(* IEC 61131-3 sources: pandora/pandora/aws-platform-main/aws-platform-main/test/Api, 3 files *)

(* ---- IoGroups.st ---- *)
USING AxUnit;

NAMESPACE Esab.Api.Test

    {TestFixture}
    CLASS DigitalOutputGroupTests
        VAR PRIVATE
            output : DigitalOutputGroup;
        END_VAR

        {FixtureSetup}
        METHOD PUBLIC TestFixtureSetup
            ;
        END_METHOD

        {TestSetup}
        METHOD PUBLIC TestSetup
            output.Output.Reset();
            output.Value := FALSE;
        END_METHOD

        {Test}
        METHOD PUBLIC MyTestMethod
            output.Output.Set();
            Assert.Equal(output.Value, FALSE);
            output.Write();
            Assert.Equal(output.Value, TRUE);

            output.Output.Reset();
            Assert.Equal(output.Value, TRUE);
            output.Write();
            Assert.Equal(output.Value, FALSE);
        END_METHOD
    END_CLASS

END_NAMESPACE

(* ---- WebApi.st ---- *)
USING Esab.Utils;
USING Esab.WeldSystem.PowerSources.Mock;
USING Esab.WeldSystem.PowerSources;
USING Esab.Motion.Mock;
USING Esab.Utils.Alarming.Mock;
USING Esab.Utils.Assets.Mock;
USING Esab.Utils.Assets;

USING AxUnit;

NAMESPACE Esab.Api.Test

    {TestFixture}
    {Category(WebApi)}
    CLASS WebApiSlideCrossTests
        VAR PRIVATE
            _api : WebApi;
            _defaultApi : WebApi;
            _webApiData : WebApiData;
            _defaultWebApiData : WebApiData;
            _horizontalSlideMock : ToPosAxisMock;
            _verticalSlideMock : ToPosAxisMock;
            _assetsManagerMock : AssetsManagerMock;
        END_VAR

        {FixtureSetup}
        METHOD PUBLIC TestFixtureSetup
            _api := _defaultApi;
            _api.Setup(_assetsManagerMock, REF(_webApiData));
        END_METHOD

        {TestSetup}
        METHOD PUBLIC TestSetup
            _webApiData := _defaultWebApiData;

            _horizontalSlideMock.MockReset();
            _verticalSlideMock.MockReset();
            _assetsManagerMock.MockReset();

            // Configure assets manager mock: by default hand out the horizontal axis when requested
            _assetsManagerMock.RequestAssetHandleMock.Qualifier := AssetIdentifier#HorizontalSlideAxis;
            _assetsManagerMock.RequestAssetHandleMock.Asset := REF(_horizontalSlideMock);
            // Observables are not required for these tests; let ObserveAsset return NULL by default
            _assetsManagerMock.ObserveAssetMock.Value := NULL;
        END_METHOD

        {Test}
        METHOD PUBLIC HorizontalSlideEnable
            _webApiData.Inputs.HorizontalSlide.Commands.Enable.Execute.Read(TRUE);

            _api.Execute();

            Assert.Equal(_horizontalSlideMock.PowerOnMock.GetCallCount(), UINT#1);
        END_METHOD

        {Test}
        METHOD PUBLIC VerticalSlideEnable
            // Reconfigure assets manager mock to return vertical axis for this test
            _assetsManagerMock.RequestAssetHandleMock.Qualifier := AssetIdentifier#VerticalSlideAxis;
            _assetsManagerMock.RequestAssetHandleMock.Asset := REF(_verticalSlideMock);

            _webApiData.Inputs.VerticalSlide.Commands.Enable.Execute.Read(TRUE);

            _api.Execute();

            Assert.Equal(_verticalSlideMock.PowerOnMock.GetCallCount(), UINT#1);
        END_METHOD

        {Test}
        METHOD PUBLIC HorizontalSlideAbsolutePositionCommand
            _webApiData.Inputs.HorizontalSlide.Commands.Positioning.CommandType.Read(PositioningCommandType#Absolute);
            _webApiData.Inputs.HorizontalSlide.Commands.Positioning.Position.Read(REAL#1.0);
            _webApiData.Inputs.HorizontalSlide.Commands.Positioning.Velocity.Read(REAL#2.0);
            _webApiData.Inputs.HorizontalSlide.Commands.Positioning.Acceleration.Read(REAL#3.0);
            _webApiData.Inputs.HorizontalSlide.Commands.Positioning.Deceleration.Read(REAL#4.0);
            _webApiData.Inputs.HorizontalSlide.Commands.Positioning.Jerk.Read(REAL#5.0);
            _webApiData.Inputs.HorizontalSlide.Commands.Positioning.Execute.Read(TRUE);

            _api.Execute();

            Assert.Equal(_horizontalSlideMock.ExecutePositioningCommandMock.GetCallCount(), UINT#1);
            //Assert.Equal(_horizontalSlideHandlerMock.ExecuteCommandMock.Command.Id, 123);
            Assert.Equal(_horizontalSlideMock.ExecutePositioningCommandMock.Command.CommandType, Esab.Motion.AxisCommandType#Absolute);
            Assert.Equal(_horizontalSlideMock.ExecutePositioningCommandMock.Command.Position, 1.0);
            Assert.Equal(_horizontalSlideMock.ExecutePositioningCommandMock.Command.Velocity, 2.0);
            Assert.Equal(_horizontalSlideMock.ExecutePositioningCommandMock.Command.Acceleration, 3.0);
            Assert.Equal(_horizontalSlideMock.ExecutePositioningCommandMock.Command.Deceleration, 4.0);
            Assert.Equal(_horizontalSlideMock.ExecutePositioningCommandMock.Command.Jerk, 5.0);
            ;
        END_METHOD

        {Test}
        METHOD PUBLIC HorizontalSlideRelativePositionCommand
            _webApiData.Inputs.HorizontalSlide.Commands.Positioning.CommandType.Read(PositioningCommandType#Relative);
            _webApiData.Inputs.HorizontalSlide.Commands.Positioning.Position.Read(REAL#1.0);
            _webApiData.Inputs.HorizontalSlide.Commands.Positioning.Velocity.Read(REAL#2.0);
            _webApiData.Inputs.HorizontalSlide.Commands.Positioning.Acceleration.Read(REAL#3.0);
            _webApiData.Inputs.HorizontalSlide.Commands.Positioning.Deceleration.Read(REAL#4.0);
            _webApiData.Inputs.HorizontalSlide.Commands.Positioning.Jerk.Read(REAL#5.0);
            _webApiData.Inputs.HorizontalSlide.Commands.Positioning.Execute.Read(TRUE);

            _api.Execute();

            Assert.Equal(_horizontalSlideMock.ExecutePositioningCommandMock.GetCallCount(), UINT#1);
            //Assert.Equal(_horizontalSlideHandlerMock.ExecuteCommandMock.Command.Id, 123);
            Assert.Equal(_horizontalSlideMock.ExecutePositioningCommandMock.Command.CommandType, Esab.Motion.AxisCommandType#Relative);
            Assert.Equal(_horizontalSlideMock.ExecutePositioningCommandMock.Command.Position, 1.0);
            Assert.Equal(_horizontalSlideMock.ExecutePositioningCommandMock.Command.Velocity, 2.0);
            Assert.Equal(_horizontalSlideMock.ExecutePositioningCommandMock.Command.Acceleration, 3.0);
            Assert.Equal(_horizontalSlideMock.ExecutePositioningCommandMock.Command.Deceleration, 4.0);
            Assert.Equal(_horizontalSlideMock.ExecutePositioningCommandMock.Command.Jerk, 5.0);
        END_METHOD

        {Test}
        METHOD PUBLIC HorizontalSlideVelocityCommand
            _webApiData.Inputs.HorizontalSlide.Commands.Positioning.CommandType.Read(PositioningCommandType#Velocity);
            _webApiData.Inputs.HorizontalSlide.Commands.Positioning.Position.Read(REAL#1.0);
            _webApiData.Inputs.HorizontalSlide.Commands.Positioning.Velocity.Read(REAL#2.0);
            _webApiData.Inputs.HorizontalSlide.Commands.Positioning.Acceleration.Read(REAL#3.0);
            _webApiData.Inputs.HorizontalSlide.Commands.Positioning.Deceleration.Read(REAL#4.0);
            _webApiData.Inputs.HorizontalSlide.Commands.Positioning.Jerk.Read(REAL#5.0);
            _webApiData.Inputs.HorizontalSlide.Commands.Positioning.Execute.Read(TRUE);

            _api.Execute();

            Assert.Equal(_horizontalSlideMock.ExecutePositioningCommandMock.GetCallCount(), UINT#1);
            //Assert.Equal(_horizontalSlideHandlerMock.ExecuteCommandMock.Command.Id, 123);
            Assert.Equal(_horizontalSlideMock.ExecutePositioningCommandMock.Command.CommandType, Esab.Motion.AxisCommandType#Velocity);
            Assert.Equal(_horizontalSlideMock.ExecutePositioningCommandMock.Command.Position, 1.0);
            Assert.Equal(_horizontalSlideMock.ExecutePositioningCommandMock.Command.Velocity, 2.0);
            Assert.Equal(_horizontalSlideMock.ExecutePositioningCommandMock.Command.Acceleration, 3.0);
            Assert.Equal(_horizontalSlideMock.ExecutePositioningCommandMock.Command.Deceleration, 4.0);
            Assert.Equal(_horizontalSlideMock.ExecutePositioningCommandMock.Command.Jerk, 5.0);
        END_METHOD

        {Test}
        METHOD PUBLIC HorizontalSlideHaltCommand
            _webApiData.Inputs.HorizontalSlide.Commands.Positioning.CommandType.Read(PositioningCommandType#Halt);
            _webApiData.Inputs.HorizontalSlide.Commands.Positioning.Position.Read(REAL#1.0);
            _webApiData.Inputs.HorizontalSlide.Commands.Positioning.Velocity.Read(REAL#2.0);
            _webApiData.Inputs.HorizontalSlide.Commands.Positioning.Acceleration.Read(REAL#3.0);
            _webApiData.Inputs.HorizontalSlide.Commands.Positioning.Deceleration.Read(REAL#4.0);
            _webApiData.Inputs.HorizontalSlide.Commands.Positioning.Jerk.Read(REAL#5.0);
            _webApiData.Inputs.HorizontalSlide.Commands.Positioning.Execute.Read(TRUE);

            _api.Execute();

            Assert.Equal(_horizontalSlideMock.ExecutePositioningCommandMock.GetCallCount(), UINT#1);
            //Assert.Equal(_horizontalSlideHandlerMock.ExecuteCommandMock.Command.Id, 123);
            Assert.Equal(_horizontalSlideMock.ExecutePositioningCommandMock.Command.CommandType, Esab.Motion.AxisCommandType#Halt);
            Assert.Equal(_horizontalSlideMock.ExecutePositioningCommandMock.Command.Position, 1.0);
            Assert.Equal(_horizontalSlideMock.ExecutePositioningCommandMock.Command.Velocity, 2.0);
            Assert.Equal(_horizontalSlideMock.ExecutePositioningCommandMock.Command.Acceleration, 3.0);
            Assert.Equal(_horizontalSlideMock.ExecutePositioningCommandMock.Command.Deceleration, 4.0);
            Assert.Equal(_horizontalSlideMock.ExecutePositioningCommandMock.Command.Jerk, 5.0);
        END_METHOD

        {Test}
        METHOD PUBLIC HorizontalSlideDirectAbsoluteHomingCommand

            _webApiData.Inputs.HorizontalSlide.Commands.Homing.HomingType.Read(HomingCommandType#DirectAbsolute);
            _webApiData.Inputs.HorizontalSlide.Commands.Homing.Position.Read(REAL#10.0);
            _webApiData.Inputs.HorizontalSlide.Commands.Homing.Execute.Read(TRUE);

            _api.Execute();

            Assert.Equal(_horizontalSlideMock.ExecuteHomingCommandMock.GetCallCount(), UINT#1);
            Assert.Equal(_horizontalSlideMock.ExecuteHomingCommandMock.Command.HomingType, Esab.Motion.AxisHomingType#DirectAbsolute);
            Assert.Equal(_horizontalSlideMock.ExecuteHomingCommandMock.Command.Position, 10.0);
        END_METHOD
    END_CLASS

    {TestFixture}
    {Category(WebApi)}
    CLASS WebApiWeldTests
        VAR PRIVATE
            _api : WebApi;
            _webApiData : WebApiData;
            _powerSourceMock : Aristo1000Mock;
            _assetsManagerMock : AssetsManagerMock;
        END_VAR

        {FixtureSetup}
        METHOD PUBLIC TestFixtureSetup
            _api.Setup(_assetsManagerMock, REF(_webApiData));
        END_METHOD

        {TestSetup}
        METHOD PUBLIC TestSetup
            THIS.ResetWebApiData();

            _powerSourceMock.MockReset();
            _assetsManagerMock.MockReset();

            _assetsManagerMock.RequestAssetHandleMock.Qualifier := AssetIdentifier#PowerSource1;
            _assetsManagerMock.RequestAssetHandleMock.Asset := REF(_powerSourceMock);
            // Observables are not required for these tests; let ObserveAsset return NULL by default
            _assetsManagerMock.ObserveAssetMock.Value := NULL;
        END_METHOD

        METHOD PRIVATE ResetWebApiData
            // Commands
            _webApiData.Inputs.PowerSource1.Commands.StartWeld.Execute.Read(FALSE);
            _webApiData.Inputs.PowerSource1.Commands.StartWeld.Execute.Read(FALSE);

            _webApiData.Inputs.PowerSource1.Commands.StopWeld.Execute.Read(FALSE);
            _webApiData.Inputs.PowerSource1.Commands.StopWeld.Execute.Read(FALSE);

            _webApiData.Inputs.PowerSource1.Commands.UpdateStatus.Execute.Read(FALSE);
            _webApiData.Inputs.PowerSource1.Commands.UpdateStatus.Execute.Read(FALSE);

            // Parameters
            _webApiData.Inputs.PowerSource1.ActiveArea.AcBalance.Read(UINT#0);
            _webApiData.Inputs.PowerSource1.ActiveArea.AcFrequency.Read(UINT#0);
            _webApiData.Inputs.PowerSource1.ActiveArea.AcOffset.Read(UINT#0);
            _webApiData.Inputs.PowerSource1.ActiveArea.AcPhaseShift.Read(UINT#0);
            _webApiData.Inputs.PowerSource1.ActiveArea.Current.Read(UINT#0);
            _webApiData.Inputs.PowerSource1.ActiveArea.IceWireSpeedPercentage.Read(UINT#0);
            _webApiData.Inputs.PowerSource1.ActiveArea.RegulationDynamics.Read(UINT#0);
            _webApiData.Inputs.PowerSource1.ActiveArea.RegulationInductance.Read(UINT#0);
            _webApiData.Inputs.PowerSource1.ActiveArea.RegulationType.Read(UINT#0);
            _webApiData.Inputs.PowerSource1.ActiveArea.StartAdjust.Read(UINT#0);
            _webApiData.Inputs.PowerSource1.ActiveArea.TravelSpeed.Read(UINT#0);
            _webApiData.Inputs.PowerSource1.ActiveArea.Voltage.Read(UINT#0);

            _webApiData.Inputs.PowerSource1.WeldDataSet.AcBalance.Read(UINT#0);
            _webApiData.Inputs.PowerSource1.WeldDataSet.AcFrequency.Read(UINT#0);
            _webApiData.Inputs.PowerSource1.WeldDataSet.AcOffset.Read(UINT#0);
            _webApiData.Inputs.PowerSource1.WeldDataSet.AcPhaseShift.Read(UINT#0);
            _webApiData.Inputs.PowerSource1.WeldDataSet.Current.Read(UINT#0);
            _webApiData.Inputs.PowerSource1.WeldDataSet.IceWireSpeedPercentage.Read(UINT#0);
            _webApiData.Inputs.PowerSource1.WeldDataSet.RegulationDynamics.Read(UINT#0);
            _webApiData.Inputs.PowerSource1.WeldDataSet.RegulationInductance.Read(UINT#0);
            _webApiData.Inputs.PowerSource1.WeldDataSet.RegulationType.Read(UINT#0);
            _webApiData.Inputs.PowerSource1.WeldDataSet.StartAdjust.Read(UINT#0);
            _webApiData.Inputs.PowerSource1.WeldDataSet.TravelSpeed.Read(UINT#0);
            _webApiData.Inputs.PowerSource1.WeldDataSet.Voltage.Read(UINT#0);
        END_METHOD

        {Test}
        METHOD PUBLIC AssetManagerMockRequestAsset
            VAR_TEMP
                asset : REF_TO Asset;
                handle : IPowerSource;
            END_VAR

            _assetsManagerMock.RequestAssetHandleMock.Qualifier := AssetIdentifier#PowerSource1;
            _assetsManagerMock.RequestAssetHandleMock.Asset := REF(_powerSourceMock);

            asset := _assetsManagerMock.RequestAssetHandle(_api, AssetIdentifier#PowerSource1);

            Assert.Equal(asset <> NULL, TRUE);

            handle ?= asset^;

            Assert.Equal(handle <> NULL, TRUE);
        END_METHOD

        {Test}
        METHOD PUBLIC PowerSource1WriteAsync
            _webApiData.Inputs.PowerSource1.Commands.WriteAsync.Index.Read(DINT#46);
            _webApiData.Inputs.PowerSource1.Commands.WriteAsync.Value.Read(UINT#2);
            _webApiData.Inputs.PowerSource1.Commands.WriteAsync.Execute.Read(TRUE);

            Assert.Equal(_powerSourceMock.WriteAsyncCmdMock.GetCallCount(), UINT#1);
            Assert.Equal(_powerSourceMock.WriteAsyncCmdMock.Command = NULL, FALSE);
            Assert.Equal(_powerSourceMock.WriteAsyncCmdMock.Command^.Index, DINT#46);
            Assert.Equal(_powerSourceMock.WriteAsyncCmdMock.Command^.Value, DINT#2);
        END_METHOD

        {Test}
        METHOD PUBLIC PowerSource1ReadAsync
            VAR_TEMP
                command : REF_TO UIntAsyncCommand := NULL;
            END_VAR
            _webApiData.Inputs.PowerSource1.Commands.ReadAsync.Index.Read(DINT#46);
            _webApiData.Inputs.PowerSource1.Commands.ReadAsync.Execute.Read(TRUE);

            Assert.Equal(_powerSourceMock.ReadAsyncCmdMock.GetCallCount(), UINT#1);
            Assert.Equal(_powerSourceMock.ReadAsyncCmdMock.Command = NULL, FALSE);
            Assert.Equal(_powerSourceMock.ReadAsyncCmdMock.Command^.Index, DINT#46);
            Assert.Equal(_webApiData.Outputs.PowerSource1.Commands.ReadAsync.Busy.Value, TRUE);
            Assert.Equal(_webApiData.Outputs.PowerSource1.Commands.ReadAsync.Executed.Value, TRUE);

            _webApiData.Inputs.PowerSource1.Commands.ReadAsync.Execute.Read(FALSE);
            Assert.Equal(_webApiData.Outputs.PowerSource1.Commands.ReadAsync.Executed.Value, FALSE);
            Assert.Equal(_webApiData.Outputs.PowerSource1.Commands.ReadAsync.Busy.Value, TRUE);

            command := _powerSourceMock.ReadAsyncCmdMock.Command;
            command^.Value := UINT#20;

            _api.AsyncCommandCallback(command, CommandStatus#Success);
            Assert.Equal(_webApiData.Outputs.PowerSource1.Commands.ReadAsync.Busy.Value, FALSE);
            Assert.Equal(_webApiData.Outputs.PowerSource1.Commands.ReadAsync.ErrorCode.Value, UINT#0);
            Assert.Equal(_webApiData.Outputs.PowerSource1.Commands.ReadAsync.Value.Value, UINT#20);
        END_METHOD

        {Test}
        METHOD PUBLIC PowerSource1ReadAsyncFailiure
            VAR_TEMP
                command : REF_TO UIntAsyncCommand := NULL;
            END_VAR
            _webApiData.Inputs.PowerSource1.Commands.ReadAsync.Index.Read(DINT#46);
            _webApiData.Inputs.PowerSource1.Commands.ReadAsync.Execute.Read(TRUE);
            _webApiData.Inputs.PowerSource1.Commands.ReadAsync.Execute.Read(FALSE);

            command := _powerSourceMock.ReadAsyncCmdMock.Command;
            command^.Value := UINT#20;

            _api.AsyncCommandCallback(command, CommandStatus#Error);
            Assert.Equal(_webApiData.Outputs.PowerSource1.Commands.ReadAsync.Busy.Value, FALSE);
            Assert.Equal(_webApiData.Outputs.PowerSource1.Commands.ReadAsync.ErrorCode.Value, UINT#2);
        END_METHOD
    END_CLASS

END_NAMESPACE

(* ---- WebApiBlock.st ---- *)
USING Esab.Api;
USING Esab.Utils.Assets;
USING Esab.Motion.Mock;
USING Esab.Motion;
USING AxUnit;

NAMESPACE Esab.Api.BlockTests

    {TestFixture}
    {Category(Blocks)}
    CLASS WebApiBlockTests
        VAR PRIVATE
            _api : WebApi;
            _image : WebApiData; // Simulated IO image with Inputs/Outputs
            _assets : AssetsManager;
            _hAxis : ToPosAxisMock;
            _hAxisObservable : REF_TO AxisObservable;
        END_VAR

        {TestSetup}
        METHOD PUBLIC Setup
            // Reset and bind API
            _hAxis.MockReset();
            _hAxisObservable ?= _hAxis.Observe();

            // Clear image values
            _image.Inputs.HorizontalSlide.Commands.Enable.Execute.Value := FALSE;
            _image.Inputs.HorizontalSlide.Commands.Disable.Execute.Value := FALSE;
            _image.Inputs.HorizontalSlide.Commands.Halt.Execute.Value := FALSE;
            _image.Inputs.HorizontalSlide.Commands.JogPositive.Execute.Value := FALSE;
            _image.Inputs.HorizontalSlide.Commands.JogNegative.Execute.Value := FALSE;
            _image.Inputs.HorizontalSlide.Commands.Positioning.Execute.Value := FALSE;
            _image.Inputs.HorizontalSlide.Commands.Positioning.CommandType.Value := UINT#0;
            _image.Inputs.HorizontalSlide.Commands.Positioning.Position.Value := REAL#0.0;
            _image.Inputs.HorizontalSlide.Commands.Positioning.Velocity.Value := REAL#0.0;
            _image.Inputs.HorizontalSlide.Commands.Positioning.Acceleration.Value := REAL#0.0;
            _image.Inputs.HorizontalSlide.Commands.Positioning.Deceleration.Value := REAL#0.0;
            _image.Inputs.HorizontalSlide.Commands.Positioning.Jerk.Value := REAL#0.0;
            _image.Inputs.HorizontalSlide.Commands.Homing.Execute.Value := FALSE;
            _image.Inputs.HorizontalSlide.Commands.Homing.HomingType.Value := UINT#0;
            _image.Inputs.HorizontalSlide.Commands.Homing.Position.Value := REAL#0.0;

            // Bind API to image and asset manager
            _api.Setup(_assets, REF(_image));

            // Register axis mocks as managed assets (block-level intent)
            // Assign identifiers so the real AssetsManager can index them
            _hAxis.SetIdentifier(AssetIdentifier#HorizontalSlideAxis);
            _assets.RegisterAsset(REF(_hAxis));
        END_METHOD

        // Helper: propagate input image values into IO classes (produce edges when toggled)
        METHOD PRIVATE PropagateInputsHorizontal
            _image.Inputs.HorizontalSlide.Commands.Enable.Execute.Read();
            _image.Inputs.HorizontalSlide.Commands.Disable.Execute.Read();
            _image.Inputs.HorizontalSlide.Commands.Halt.Execute.Read();
            _image.Inputs.HorizontalSlide.Commands.JogPositive.Execute.Read();
            _image.Inputs.HorizontalSlide.Commands.JogNegative.Execute.Read();

            _image.Inputs.HorizontalSlide.Commands.Positioning.CommandType.Read();
            _image.Inputs.HorizontalSlide.Commands.Positioning.Position.Read();
            _image.Inputs.HorizontalSlide.Commands.Positioning.Velocity.Read();
            _image.Inputs.HorizontalSlide.Commands.Positioning.Acceleration.Read();
            _image.Inputs.HorizontalSlide.Commands.Positioning.Deceleration.Read();
            _image.Inputs.HorizontalSlide.Commands.Positioning.Jerk.Read();
            _image.Inputs.HorizontalSlide.Commands.Positioning.Execute.Read();

            _image.Inputs.HorizontalSlide.Commands.Homing.HomingType.Read();
            _image.Inputs.HorizontalSlide.Commands.Homing.Position.Read();
            _image.Inputs.HorizontalSlide.Commands.Homing.Execute.Read();
        END_METHOD

        METHOD PRIVATE Execute
            THIS.PropagateInputsHorizontal();
            _api.Execute();
            THIS.PropagateOutputsHorizontal();
        END_METHOD

        METHOD PRIVATE PropagateOutputsHorizontal
            _image.Outputs.HorizontalSlide.Valid.Write();
            _image.Outputs.HorizontalSlide.Status.Enabled.Write();
            _image.Outputs.HorizontalSlide.Status.Homed.Write();
            _image.Outputs.HorizontalSlide.Status.Error.Write();
            _image.Outputs.HorizontalSlide.Status.Busy.Write();
            _image.Outputs.HorizontalSlide.Status.Position.Write();
            _image.Outputs.HorizontalSlide.Status.Velocity.Write();
        END_METHOD

        // Test: Positioning command absolute on horizontal axis via IO image and observable mapping
        {Test}
        METHOD PUBLIC Horizontal_PositionAbsolute_UpdatesAxisAndOutputs
            // 1) Prime edges low
            _image.Inputs.HorizontalSlide.Commands.Positioning.Execute.Value := FALSE;
            THIS.Execute();

            // 2) Set up parameters and rising edge for execute
            _image.Inputs.HorizontalSlide.Commands.Positioning.CommandType.Value := PositioningCommandType#Absolute;
            _image.Inputs.HorizontalSlide.Commands.Positioning.Position.Value := REAL#12.5;
            _image.Inputs.HorizontalSlide.Commands.Positioning.Velocity.Value := REAL#2.5;
            _image.Inputs.HorizontalSlide.Commands.Positioning.Acceleration.Value := REAL#3.5;
            _image.Inputs.HorizontalSlide.Commands.Positioning.Deceleration.Value := REAL#4.5;
            _image.Inputs.HorizontalSlide.Commands.Positioning.Jerk.Value := REAL#5.5;
            _image.Inputs.HorizontalSlide.Commands.Positioning.Execute.Value := TRUE; // Rising

            // Drive to test outputs mapping
            _hAxis.IsEnabledMock.Value := TRUE;
            _hAxis.IsHomedMock.Value := TRUE;
            _hAxis.HasErrorMock.Value := FALSE;
            _hAxis.IsBusyMock.Value := TRUE;
            _hAxis.ActualLinearPositionMock.Value := LREAL#12.5;
            _hAxis.ActualLinearVelocityMock.Value := LREAL#2.5;

            THIS.Execute();

            // Verify command reached axis (through observable mock’s recorded command)
            Assert.Equal(_hAxis.ExecutePositioningCommandMock.GetCallCount(), UINT#1);

            Assert.Equal(_hAxis.ExecutePositioningCommandMock.Command.CommandType, Esab.Motion.AxisCommandType#Absolute);
            Assert.Equal(_hAxis.ExecutePositioningCommandMock.Command.Position, 12.5);
            Assert.Equal(_hAxis.ExecutePositioningCommandMock.Command.Velocity, 2.5);
        END_METHOD

        // Test: Homing command on Horizontal axis
        {Test}
        METHOD PUBLIC Horizontal_HomingDirectAbsolute_UpdatesAxis
            // AssetsManager is real; horizontal axis is already registered with correct ID.

            // Prime low then rise
            _image.Inputs.HorizontalSlide.Commands.Homing.Execute.Value := FALSE;
            THIS.Execute();

            _image.Inputs.HorizontalSlide.Commands.Homing.HomingType.Value := HomingCommandType#DirectAbsolute;
            _image.Inputs.HorizontalSlide.Commands.Homing.Position.Value := REAL#10.0;
            _image.Inputs.HorizontalSlide.Commands.Homing.Execute.Value := TRUE;

            THIS.Execute();

            Assert.Equal(_hAxis.ExecuteHomingCommandMock.GetCallCount(), UINT#1);
            Assert.Equal(_hAxis.ExecuteHomingCommandMock.Command.HomingType, Esab.Motion.AxisHomingType#DirectAbsolute);
            Assert.Equal(_hAxis.ExecuteHomingCommandMock.Command.Position, 10.0);
        END_METHOD

        // Test: Enable command on horizontal axis using Value+Read propagation toggling
        {Test}
        METHOD PUBLIC Horizontal_Enable_TogglesOnce
            // Use horizontal axis (mock with PowerOnMock) to verify enable edge behavior
            // Prime low
            _image.Inputs.HorizontalSlide.Commands.Enable.Execute.Value := FALSE;
            THIS.Execute();
            Assert.Equal(_hAxis.PowerOnMock.GetCallCount(), UINT#0);

            // Set high and propagate
            _image.Inputs.HorizontalSlide.Commands.Enable.Execute.Value := TRUE;
            THIS.Execute();
            Assert.Equal(_image.Inputs.HorizontalSlide.Commands.Enable.Execute.Value, FALSE);

            Assert.Equal(_hAxis.PowerOnMock.GetCallCount(), UINT#1);
        END_METHOD

        // Test: Axis remains locked while Busy across cycles
        {Test}
        METHOD PUBLIC Horizontal_PositionCommand_KeepsLockWhileBusy
            VAR_TEMP
                handleAttempt : REF_TO Asset;
                cycles : UINT;
            END_VAR

            // Prime low, execute once
            _image.Inputs.HorizontalSlide.Commands.Positioning.Execute.Value := FALSE;
            THIS.Execute();

            // Issue absolute move on rising edge
            _image.Inputs.HorizontalSlide.Commands.Positioning.CommandType.Value := PositioningCommandType#Absolute;
            _image.Inputs.HorizontalSlide.Commands.Positioning.Position.Value := REAL#5.0;
            _image.Inputs.HorizontalSlide.Commands.Positioning.Velocity.Value := REAL#1.0;
            _image.Inputs.HorizontalSlide.Commands.Positioning.Acceleration.Value := REAL#2.0;
            _image.Inputs.HorizontalSlide.Commands.Positioning.Deceleration.Value := REAL#3.0;
            _image.Inputs.HorizontalSlide.Commands.Positioning.Jerk.Value := REAL#4.0;
            _image.Inputs.HorizontalSlide.Commands.Positioning.Execute.Value := TRUE;

            // Simulate multi-cycle busy
            _hAxis.IsBusyMock.Value := TRUE;

            THIS.Execute();

            // For several cycles, the asset should remain locked so that RequestAssetHandle returns NULL
            FOR cycles := UINT#0 TO UINT#2 DO
                THIS.Execute();
                handleAttempt := _assets.RequestAssetHandle(_api, AssetIdentifier#HorizontalSlideAxis);
                Assert.Equal(handleAttempt = NULL, TRUE);
            END_FOR;

            // Now mark command done/busy false and execute once to allow unlock
            _hAxis.IsBusyMock.Value := FALSE;
            THIS.Execute();

            // After Busy clears, asset should be unlocked and available
            handleAttempt := _assets.RequestAssetHandle(_api, AssetIdentifier#HorizontalSlideAxis);
            Assert.Equal(handleAttempt <> NULL, TRUE);
        END_METHOD
    END_CLASS
END_NAMESPACE
